FUNCTION_BLOCK NOT_BOOL (* IEC 61131-3 Boolean NOT *)
  (* Standard: 61131-3 *)
  (* Version 0.1, 2006-09-07, JHC, Holobloc Inc, Converted to Template *)
  (* Version 0.0, 2004-12-15, JHC, Rockwell Automation, Converted from SRC format. *)
  (* Compiler header: package fb.rt.plc.bits; *)
  (* Compiler classdef: (! in) *)
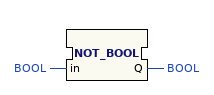
  VAR_INPUT
    in : BOOL;
  END_VAR
  VAR_OUTPUT
    Q : BOOL;
  END_VAR
END_FUNCTION_BLOCK
